DATA_BLOCK "TASK"
{ S7_Optimized_Access := 'FALSE' }
VERSION : 0.1
   STRUCT
      Status { ExternalWritable := 'False'; S7_SetPoint := 'False'} : "LGR_Equip_TaskStatus";
      Proc { ExternalWritable := 'False'; S7_SetPoint := 'False'} : "LGR_Proc_component";
      ProcBuff { ExternalWritable := 'False'; S7_SetPoint := 'False'} : "LGR_Proc_component";
      Now { ExternalWritable := 'False'; S7_SetPoint := 'False'} : "LGR_Task_Data";
      NowBuff : "LGR_Task_Data";
      Buff { ExternalWritable := 'False'; S7_SetPoint := 'False'} : Array[0..3] of "LGR_Task_Data";
      Last { ExternalWritable := 'False'; S7_SetPoint := 'False'} : Array[0..9] of "LGR_Task_Data";
      Canceled : Array[0..9] of "LGR_Task_Data";
      Rejected : Array[0..9] of "LGR_Task_Data";
      ErrorOccuredData : Struct
         Last : Array[0..9] of "LGR_Task_Data";
         Now : Array[0..9] of "LGR_Task_Data";
         Next : Array[0..9] of "LGR_Task_Data";
         "Time" {InstructionName := 'DTL'; LibVersion := '1.0'; S7_SetPoint := 'True'} : Array[0..9] of DTL;
      END_STRUCT;
      CompletePending : "LGR_Task_Data";   //    수동 완료 CV 인계 대기 작업 (Buff[0] 과 같을 때만 유효, CL_Common_Command)
      GripPassed : "LGR_Task_Data";   //    Grip(500) 을 지난 작업 - 수동 Complete 조건 (Buff[0] 과 같을 때만, PL_Task_V2)
   END_STRUCT;


BEGIN
   Proc.ProcNo := 20;

END_DATA_BLOCK

